// TwinCAT 3 PLC project Untitled1
// ProgramVersion: 3.1.4024.0
// libraries:
//   Tc2_Standard, * (Beckhoff Automation GmbH)
//   Tc2_System, * (Beckhoff Automation GmbH)
//   Tc3_Module, * (Beckhoff Automation GmbH)
// project tree:
//   / PlcTask.TcTTO
//   POUs/ FB_Child.TcPOU, FB_Parent.TcPOU, MAIN.TcPOU
// real-time tasks:
//   TASK PlcTask: cycle T#10ms, priority 20, ADS port 350

CONFIGURATION Untitled1
    RESOURCE PLC ON TwinCAT3
        TASK PlcTask(INTERVAL := T#10ms, PRIORITY := 20);
        PROGRAM MAIN WITH PlcTask : MAIN;
    END_RESOURCE
END_CONFIGURATION

// ---- POUs/MAIN.TcPOU
PROGRAM MAIN
VAR
	fb_child : FB_Child;
END_VAR

END_PROGRAM

// ---- POUs/FB_Child.TcPOU
FUNCTION_BLOCK FB_Child EXTENDS FB_Parent
VAR_INPUT
END_VAR
VAR_OUTPUT
END_VAR
VAR
END_VAR

METHOD FB_init : BOOL
VAR_INPUT
	bInitRetains : BOOL; // if TRUE, the retain variables are initialized (warm start / cold start)
	bInCopyCode : BOOL;  // if TRUE, the instance afterwards gets moved into the copy code (online change)
END_VAR
SUPER^.ref_child REF= THIS^;
END_METHOD

END_FUNCTION_BLOCK

// ---- POUs/FB_Parent.TcPOU
FUNCTION_BLOCK FB_Parent
VAR_INPUT
END_VAR
VAR_OUTPUT
END_VAR
VAR
	ref_child : REFERENCE TO FB_Child;
END_VAR

END_FUNCTION_BLOCK
